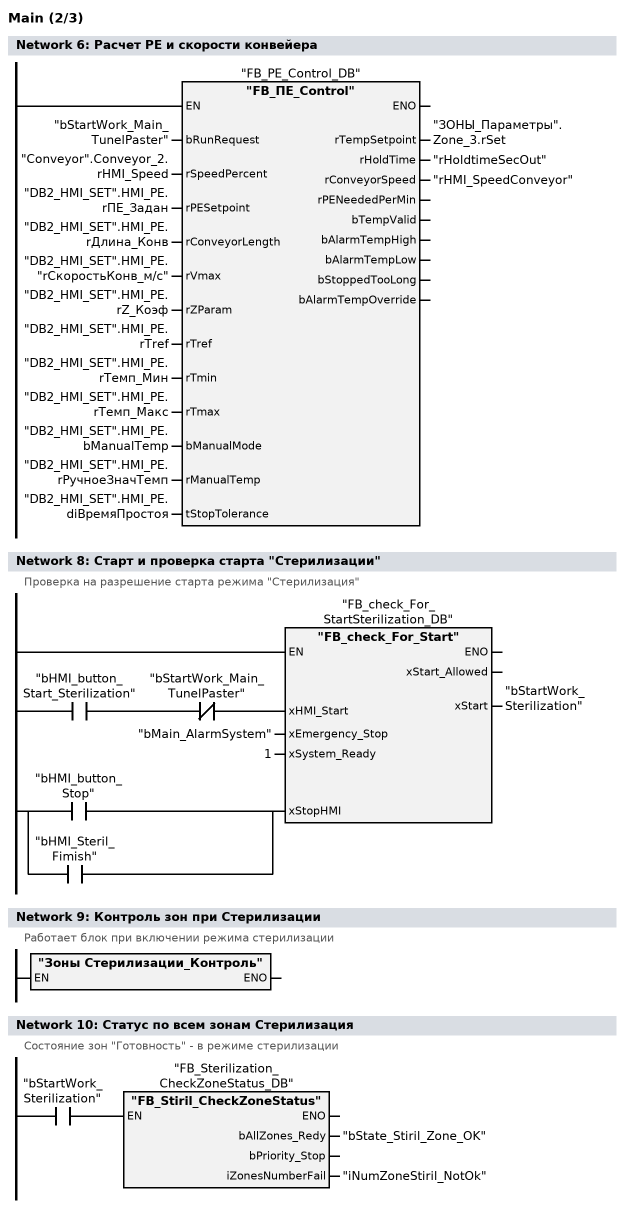
   RUNG wire#powerrail
      "FB_PE_Control_DB"(bRunRequest := "bStartWork_Main_TunelPaster", rSpeedPercent := "Conveyor".Conveyor_2.rHMI_Speed, rPESetpoint := "DB2_HMI_SET".HMI_PE.rПЕ_Задан, rConveyorLength := "DB2_HMI_SET".HMI_PE.rДлина_Конв, rVmax := "DB2_HMI_SET".HMI_PE."rСкоростьКонв_м/с", rZParam := "DB2_HMI_SET".HMI_PE.rZ_Коэф, rTref := "DB2_HMI_SET".HMI_PE.rТref, rTmin := "DB2_HMI_SET".HMI_PE.rТемп_Мин, rTmax := "DB2_HMI_SET".HMI_PE.rТемп_Макс, bManualMode := "DB2_HMI_SET".HMI_PE.bManualTemp, rManualTemp := "DB2_HMI_SET".HMI_PE.rРучноеЗначТемп, tStopTolerance := "DB2_HMI_SET".HMI_PE.diВремяПростоя, rTempSetpoint => "ЗОНЫ_Параметры".Zone_3.rSet, rHoldTime => "rHoldtimeSecOut", rConveyorSpeed => "rHMI_SpeedConveyor", rPENeededPerMin =>, bTempValid =>, bAlarmTempHigh =>, bAlarmTempLow =>, bStoppedTooLong =>, bAlarmTempOverride =>)
   END_RUNG
   // the same network as SCL:
   "FB_PE_Control_DB"(bRunRequest := "bStartWork_Main_TunelPaster",   // "FB_ПЕ_Control"
                      rSpeedPercent := "Conveyor".Conveyor_2.rHMI_Speed,
                      rPESetpoint := "DB2_HMI_SET".HMI_PE.rПЕ_Задан,
                      rConveyorLength := "DB2_HMI_SET".HMI_PE.rДлина_Конв,
                      rVmax := "DB2_HMI_SET".HMI_PE."rСкоростьКонв_м/с",
                      rZParam := "DB2_HMI_SET".HMI_PE.rZ_Коэф,
                      rTref := "DB2_HMI_SET".HMI_PE.rТref,
                      rTmin := "DB2_HMI_SET".HMI_PE.rТемп_Мин,
                      rTmax := "DB2_HMI_SET".HMI_PE.rТемп_Макс,
                      bManualMode := "DB2_HMI_SET".HMI_PE.bManualTemp,
                      rManualTemp := "DB2_HMI_SET".HMI_PE.rРучноеЗначТемп,
                      tStopTolerance := "DB2_HMI_SET".HMI_PE.diВремяПростоя,
                      rTempSetpoint => "ЗОНЫ_Параметры".Zone_3.rSet,
                      rHoldTime => "rHoldtimeSecOut",
                      rConveyorSpeed => "rHMI_SpeedConveyor");
END_REGION

REGION Network 7 (SCL): Перевод времени выдержки в минуты
   "rHMI_TimeHoldMin"  := "rHoldtimeSecOut" / 1;
   "rHMI_SpeedConveyor" := "rHMI_SpeedConveyor" * 1;
END_REGION

REGION Network 8: Старт и проверка старта "Стерилизации"
   // Проверка на разрешение старта режима "Стерилизация"
   RUNG wire#powerrail
      "FB_check_For_StartSterilization_DB"(xHMI_Start := wire#w1, xStopHMI := wire#w2, xEmergency_Stop := "bMain_AlarmSystem", xSystem_Ready := 1, xStart_Allowed =>, xStart => "bStartWork_Sterilization")
   END_RUNG
   RUNG wire#powerrail
      Contact( "bHMI_button_Start_Sterilization" )
      I_Contact( "bStartWork_Main_TunelPaster" )
   END_RUNG wire#w1
   RUNG wire#powerrail
      Contact( "bHMI_button_Stop" )
   END_RUNG wire#w2
   RUNG wire#powerrail
      Contact( "bHMI_Steril_Fimish" )
   END_RUNG wire#w2
   // the same network as SCL:
   "FB_check_For_StartSterilization_DB"(xHMI_Start := "bHMI_button_Start_Sterilization" AND NOT "bStartWork_Main_TunelPaster",   // "FB_check_For_Start"
                           xEmergency_Stop := "bMain_AlarmSystem",
                           xSystem_Ready := 1,
                           xStopHMI := "bHMI_button_Stop" OR "bHMI_Steril_Fimish",
                           xStart => "bStartWork_Sterilization");
END_REGION

REGION Network 9: Контроль зон при Стерилизации
   // Работает блок при включении режима стерилизации
   RUNG wire#powerrail
      "Зоны Стерилизации_Контроль"()
   END_RUNG
   // the same network as SCL:
   "Зоны Стерилизации_Контроль"();
END_REGION

REGION Network 10: Статус по всем зонам Стерилизация
   // Состояние зон "Готовность" - в режиме стерилизации
   RUNG wire#powerrail
      Contact( "bStartWork_Sterilization" )
      "FB_Sterilization_CheckZoneStatus_DB"(bAllZones_Redy => "bState_Stiril_Zone_OK", bPriority_Stop =>, iZonesNumberFail => "iNumZoneStiril_NotOk")
   END_RUNG
   // the same network as SCL:
   IF "bStartWork_Sterilization" THEN
       "FB_Sterilization_CheckZoneStatus_DB"(bAllZones_Redy => "bState_Stiril_Zone_OK",   // "FB_Stiril_CheckZoneStatus"
                               iZonesNumberFail => "iNumZoneStiril_NotOk");
   END_IF;
END_REGION

REGION Network 11: Таймер стерилизации
   // Отсчет времени стерилизации
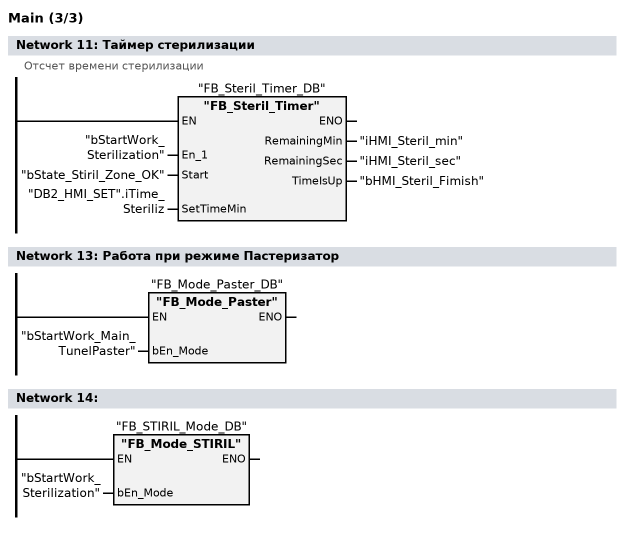
   RUNG wire#powerrail
      "FB_Steril_Timer_DB"(En_1 := "bStartWork_Sterilization", Start := "bState_Stiril_Zone_OK", SetTimeMin := "DB2_HMI_SET".iTime_Steriliz, RemainingMin => "iHMI_Steril_min", RemainingSec => "iHMI_Steril_sec", TimeIsUp => "bHMI_Steril_Fimish")
   END_RUNG
   // the same network as SCL:
   "FB_Steril_Timer_DB"(En_1 := "bStartWork_Sterilization",   // "FB_Steril_Timer"
                        Start := "bState_Stiril_Zone_OK",
                        SetTimeMin := "DB2_HMI_SET".iTime_Steriliz,
                        RemainingMin => "iHMI_Steril_min",
                        RemainingSec => "iHMI_Steril_sec",
                        TimeIsUp => "bHMI_Steril_Fimish");
END_REGION

REGION Network 12 (SCL): Окно окончания стирилизации
   IF "bHMI_Steril_Fimish" THEN
       "iHMIWind_FinishStiril" := 148;
   END_IF;
END_REGION

REGION Network 13: Работа при режиме Пастеризатор
   RUNG wire#powerrail
      "FB_Mode_Paster_DB"(bEn_Mode := "bStartWork_Main_TunelPaster")
   END_RUNG
   // the same network as SCL:
   "FB_Mode_Paster_DB"(bEn_Mode := "bStartWork_Main_TunelPaster");   // "FB_Mode_Paster"
END_REGION

REGION Network 14
   RUNG wire#powerrail
      "FB_STIRIL_Mode_DB"(bEn_Mode := "bStartWork_Sterilization")
   END_RUNG
   // the same network as SCL:
   "FB_STIRIL_Mode_DB"(bEn_Mode := "bStartWork_Sterilization");   // "FB_Mode_STIRIL"
END_REGION
END_ORGANIZATION_BLOCK

ORGANIZATION_BLOCK "PID"   // OB30, LAD, CyclicInterrupt
{ S7_Optimized_Access := 'TRUE' }
VERSION : 0.1
   VAR_INPUT
      Initial_Call : Bool;   // Initial call of this OB
      Event_Count : Int;   // Events discarded
   END_VAR
BEGIN

REGION Network 1: ПИД - Зона 1
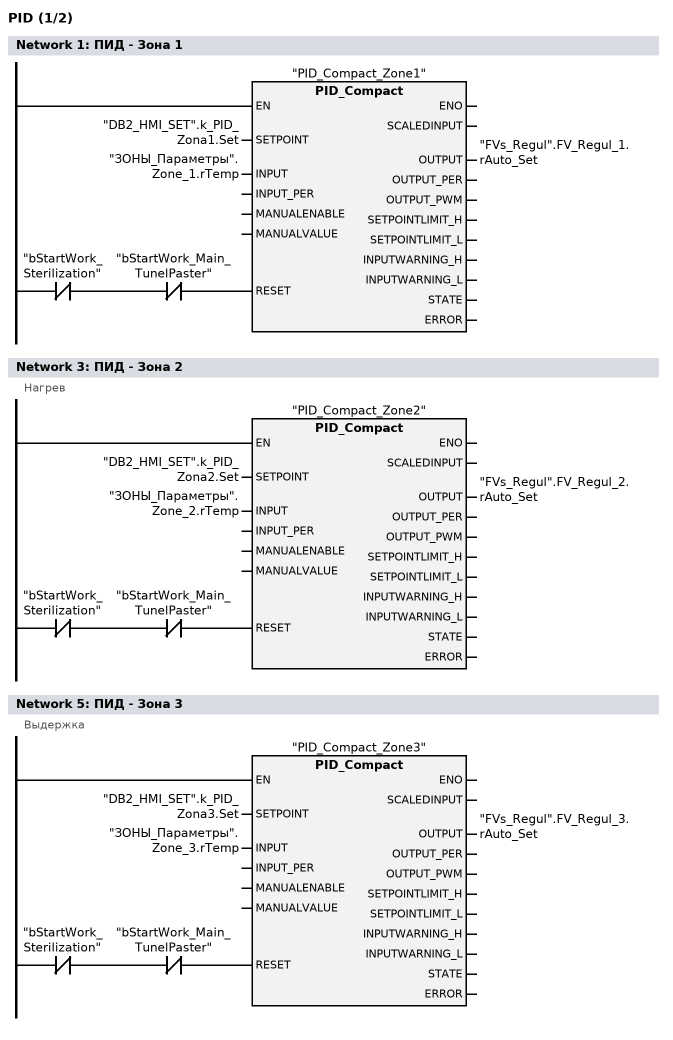
   "PID_Compact_Zone1"(Setpoint := "DB2_HMI_SET".k_PID_Zona1.Set,   // PID_Compact
                       Input := "ЗОНЫ_Параметры".Zone_1.rTemp,
                       Reset := NOT "bStartWork_Sterilization" AND NOT "bStartWork_Main_TunelPaster",
                       Output => "FVs_Regul".FV_Regul_1.rAuto_Set);
END_REGION

REGION Network 2 (SCL): Выбор типа ПИД - Зона 1
   //Режим работы ПИД - 0 - Нагрев; 1 - Охлаждение
   "PID_Compact_Zone1".sPid_Cmpt.b_InvCtrl := "bTypePID_Zone1";
   //Задание коэффициэнтов в ручном режиме

   "PID_Compact_Zone1".sRet.r_Ctrl_Gain := "DB2_HMI_SET".k_PID_Zona1.Gain; // Изменение коэф. П
   "PID_Compact_Zone1".sRet.r_Ctrl_Ti  := "DB2_HMI_SET".k_PID_Zona1.I; // Изменение коэф И
   "PID_Compact_Zone1".sRet.r_Ctrl_Td  := "DB2_HMI_SET".k_PID_Zona1.D; // Изменение коэф Д
END_REGION

REGION Network 3: ПИД - Зона 2
   // Нагрев
   "PID_Compact_Zone2"(Setpoint := "DB2_HMI_SET".k_PID_Zona2.Set,   // PID_Compact
                       Input := "ЗОНЫ_Параметры".Zone_2.rTemp,
                       Reset := NOT "bStartWork_Sterilization" AND NOT "bStartWork_Main_TunelPaster",
                       Output => "FVs_Regul".FV_Regul_2.rAuto_Set);
END_REGION

REGION Network 4 (SCL): Выбор типа ПИД Зона 2
   // 0 - Нагрев; 1 - Охлаждение
   "PID_Compact_Zone2".sPid_Cmpt.b_InvCtrl := "bTypePID_Zone2";
   //Задание коэффициэнтов в ручном режиме

   "PID_Compact_Zone2".sRet.r_Ctrl_Gain := "DB2_HMI_SET".k_PID_Zona2.Gain; // Изменение коэф. П
   "PID_Compact_Zone2".sRet.r_Ctrl_Ti := "DB2_HMI_SET".k_PID_Zona2.I; // Изменение коэф И
   "PID_Compact_Zone2".sRet.r_Ctrl_Td := "DB2_HMI_SET".k_PID_Zona2.D; // Изменение коэф Д
END_REGION

REGION Network 5: ПИД - Зона 3
   // Выдержка
   "PID_Compact_Zone3"(Setpoint := "DB2_HMI_SET".k_PID_Zona3.Set,   // PID_Compact
                       Input := "ЗОНЫ_Параметры".Zone_3.rTemp,
                       Reset := NOT "bStartWork_Sterilization" AND NOT "bStartWork_Main_TunelPaster",
                       Output => "FVs_Regul".FV_Regul_3.rAuto_Set);
END_REGION

REGION Network 6 (SCL): Выбор типа ПИД Зона 3
   // 0 - Нагрев; 1 - Охлаждение
   "PID_Compact_Zone3".sPid_Cmpt.b_InvCtrl := "bTypePID_Zone3";
   //Задание коэффициэнтов в ручном режиме
   "PID_Compact_Zone3".sRet.r_Ctrl_Gain := "DB2_HMI_SET".k_PID_Zona3.Gain; // Изменение коэф. П
   "PID_Compact_Zone3".sRet.r_Ctrl_Ti :=   "DB2_HMI_SET".k_PID_Zona3.I;    // Изменение коэф И
   "PID_Compact_Zone3".sRet.r_Ctrl_Td :=   "DB2_HMI_SET".k_PID_Zona3.D;    // Изменение коэф Д
END_REGION

REGION Network 7: ПИД - Зона 4
   // Выдержка
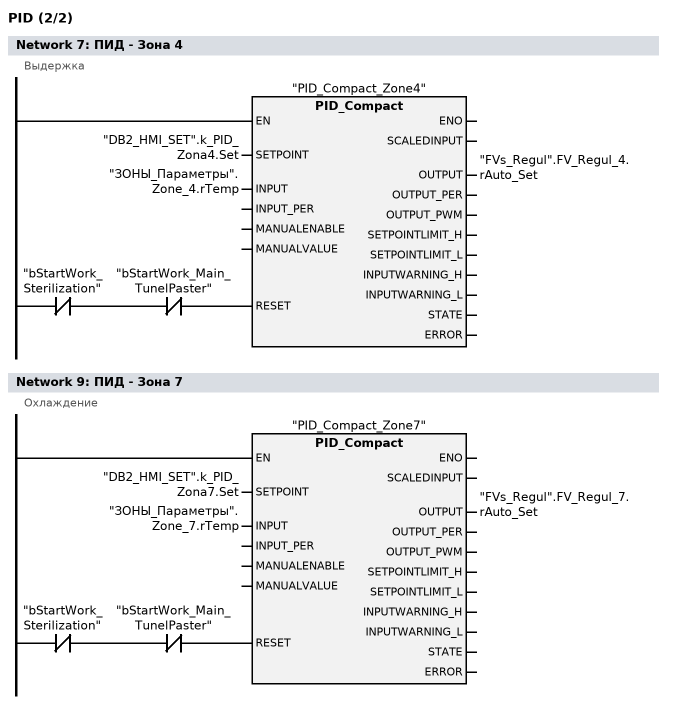
   "PID_Compact_Zone4"(Setpoint := "DB2_HMI_SET".k_PID_Zona4.Set,   // PID_Compact
                       Input := "ЗОНЫ_Параметры".Zone_4.rTemp,
                       Reset := NOT "bStartWork_Sterilization" AND NOT "bStartWork_Main_TunelPaster",
                       Output => "FVs_Regul".FV_Regul_4.rAuto_Set);
END_REGION

REGION Network 8 (SCL): Выбор типа ПИД Зона 4
   // 0 - Нагрев; 1 - Охлаждение
   "PID_Compact_Zone4".sPid_Cmpt.b_InvCtrl := TRUE;
   //Задание коэффициэнтов в ручном режиме
   "PID_Compact_Zone4".sRet.r_Ctrl_Gain := "DB2_HMI_SET".k_PID_Zona4.Gain; // Изменение коэф. П
   "PID_Compact_Zone4".sRet.r_Ctrl_Ti := "DB2_HMI_SET".k_PID_Zona4.I;    // Изменение коэф И
   "PID_Compact_Zone4".sRet.r_Ctrl_Td := "DB2_HMI_SET".k_PID_Zona4.D;    // Изменение коэф Д
END_REGION

REGION Network 9: ПИД - Зона 7
   // Охлаждение
   "PID_Compact_Zone7"(Setpoint := "DB2_HMI_SET".k_PID_Zona7.Set,   // PID_Compact
                       Input := "ЗОНЫ_Параметры".Zone_7.rTemp,
                       Reset := NOT "bStartWork_Sterilization" AND NOT "bStartWork_Main_TunelPaster",
                       Output => "FVs_Regul".FV_Regul_7.rAuto_Set);
END_REGION

REGION Network 10 (SCL): Выбор типа ПИД Зона 7
   // 0 - Нагрев; 1 - Охлаждение
   "PID_Compact_Zone7".sPid_Cmpt.b_InvCtrl := TRUE;
   //Задание коэффициэнтов в ручном режиме
   "PID_Compact_Zone7".sRet.r_Ctrl_Gain := "DB2_HMI_SET".k_PID_Zona7.Gain; // Изменение коэф. П
   "PID_Compact_Zone7".sRet.r_Ctrl_Ti := "DB2_HMI_SET".k_PID_Zona7.I;      // Изменение коэф И
   "PID_Compact_Zone7".sRet.r_Ctrl_Td := "DB2_HMI_SET".k_PID_Zona7.D;      // Изменение коэф Д
END_REGION
END_ORGANIZATION_BLOCK

ORGANIZATION_BLOCK "Startup"   // OB100, SCL, Startup
TITLE = "Complete Restart"
{ S7_Optimized_Access := 'TRUE' }
VERSION : 0.1
   VAR_INPUT
      LostRetentive : Bool;   // True if retentive data are lost
      LostRTC : Bool;   // True if date and time are lost
   END_VAR
BEGIN
   "PID_Compact_Zone1".sRet.r_Ctrl_Gain := "PID_Compact_Zone1".sBackUp.r_Gain;
END_ORGANIZATION_BLOCK

ORGANIZATION_BLOCK "Исполнительные устройств"   // OB123, LAD, ProgramCycle
TITLE = Работа физических устройств
{ S7_Optimized_Access := 'TRUE' }
VERSION : 0.1
// Насосы, клапана, и т.д.
   VAR_INPUT
      Initial_Call : Bool;   // Initial call of this OB
      Remanence : Bool;   // =True, if remanent data are available
   END_VAR
BEGIN

REGION Network 1: Аналогвые датчики
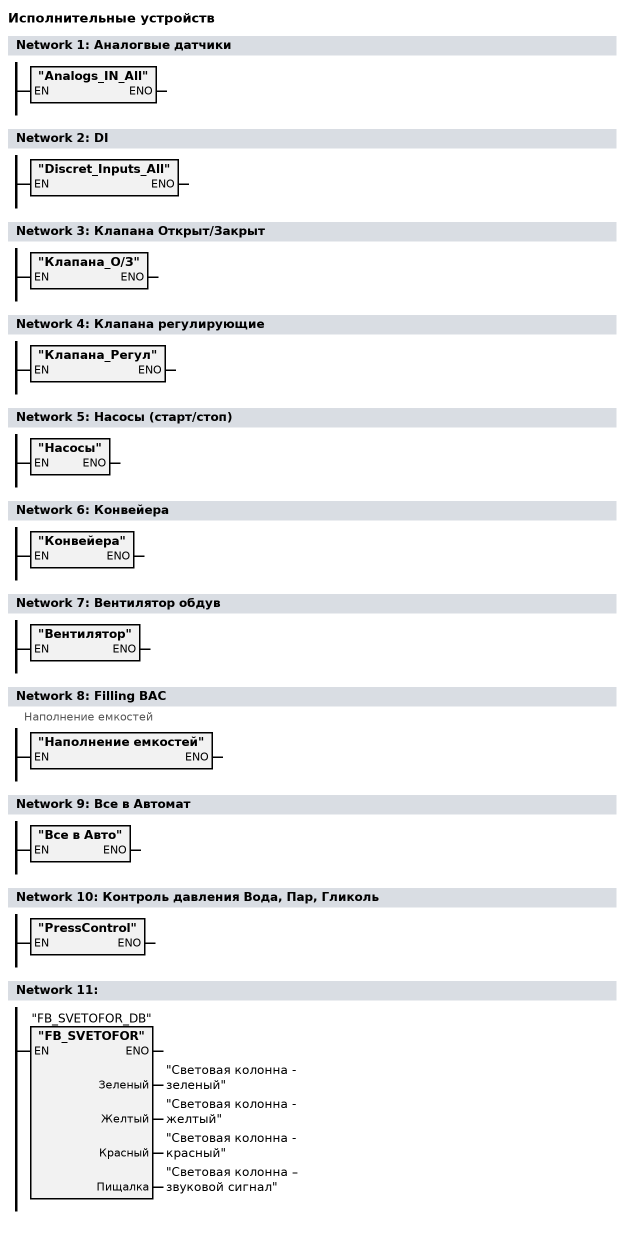
   RUNG wire#powerrail
      "Analogs_IN_All"()
   END_RUNG
   // the same network as SCL:
   "Analogs_IN_All"();
END_REGION

REGION Network 2: DI
   RUNG wire#powerrail
      "Discret_Inputs_All"()
   END_RUNG
   // the same network as SCL:
   "Discret_Inputs_All"();
END_REGION

REGION Network 3: Клапана Открыт/Закрыт
   RUNG wire#powerrail
      "Клапана_О/З"()
   END_RUNG
   // the same network as SCL:
   "Клапана_О/З"();
END_REGION

REGION Network 4: Клапана регулирующие
   RUNG wire#powerrail
      "Клапана_Регул"()
   END_RUNG
   // the same network as SCL:
   "Клапана_Регул"();
END_REGION

REGION Network 5: Насосы (старт/стоп)
   RUNG wire#powerrail
      "Насосы"()
   END_RUNG
   // the same network as SCL:
   "Насосы"();
END_REGION

REGION Network 6: Конвейера
   RUNG wire#powerrail
      "Конвейера"()
   END_RUNG
   // the same network as SCL:
   "Конвейера"();
END_REGION

REGION Network 7: Вентилятор обдув
   RUNG wire#powerrail
      "Вентилятор"()
   END_RUNG
   // the same network as SCL:
   "Вентилятор"();
END_REGION

REGION Network 8: Filling BAC
   // Наполнение емкостей
   RUNG wire#powerrail
      "Наполнение емкостей"()
   END_RUNG
   // the same network as SCL:
   "Наполнение емкостей"();
END_REGION

REGION Network 9: Все в Автомат
   RUNG wire#powerrail
      "Все в Авто"()
   END_RUNG
   // the same network as SCL:
   "Все в Авто"();
END_REGION

REGION Network 10: Контроль давления Вода, Пар, Гликоль
   RUNG wire#powerrail
      "PressControl"()
   END_RUNG
   // the same network as SCL:
   "PressControl"();
END_REGION

REGION Network 11
   RUNG wire#powerrail
      "FB_SVETOFOR_DB"(Зеленый => "Световая колонна - зеленый", Желтый => "Световая колонна - желтый", Красный => "Световая колонна - красный", Пищалка => "Световая колонна – звуковой сигнал")
   END_RUNG
   // the same network as SCL:
   "FB_SVETOFOR_DB"(Зеленый => "Световая колонна - зеленый",   // "FB_SVETOFOR"
                    Желтый => "Световая колонна - желтый",
                    Красный => "Световая колонна - красный",
                    Пищалка => "Световая колонна – звуковой сигнал");
END_REGION
END_ORGANIZATION_BLOCK

// folder: AI_Signal

FUNCTION_BLOCK "AI_(4-20)_1"   // FB13, LAD
{ S7_Optimized_Access := 'FALSE' }
VERSION : 0.1
   VAR_INPUT
      Input_PLC : Int;   // Вход_Значение на ПЛК
      "HMI_Simulate_on/off" : Bool;   // 0 - выкл, 1 - вкл
      HMI_rSimulate_value : Real;   // значение
      HMI_rParam_Sensor_HL : Real := 16.0;   // Параметры датчика по паспорту (макс значение)bar, C, итд
      HMI_rParam_Sensor_LL : Real;   // Параметры датчика по паспорту (мин значение)bar, C, итд
      "HMI_Filtr_On/off" : Bool;   // Фильтрация, true - вкл
   END_VAR
   VAR_OUTPUT
      Error_out : Bool;   // Ошибка датчика
      HMI_Value_OUT : Real;   // Значение в ед. измерения
   END_VAR
   VAR
      OUT_Scale : Real;   // Выход скалированного значения
      OUT_Normal_Ed : Real;   // Выход нормализованной единицы от 0 др 1
      AI_filtr : "AI_Filtr";
      HMI_Range : Int := 10;   // Кол-во данных для фильтрации
      HMI_iSet_Tik : Int := 2;   // Скорость набора данных для фильтрации
   END_VAR
   VAR_TEMP
      Input_PLC_to_dint : DInt;   // Конвертация из инт в реал
      Error : Word;   // Ошибка в скалировании
      "PLC to_real" : Real;
      value_scale : Real;
      Input_PLC_temp : Int;
      OFF_Param : Bool;
   END_VAR
BEGIN

REGION Network 1
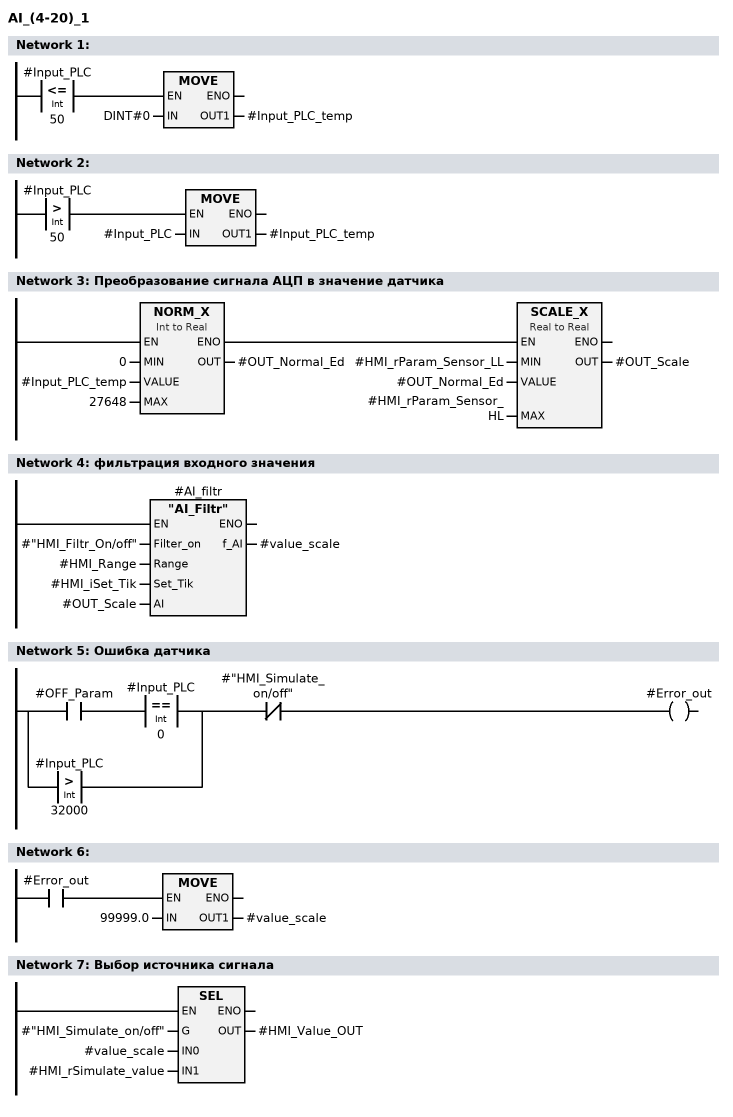
   RUNG wire#powerrail
      { S7_Templates := "SrcType := Int" } LE_Contact(in1 := #Input_PLC, in2 := 50)
      { S7_GenerateENO := "TRUE" } Move(in := DINT#0, out1 => #Input_PLC_temp)
   END_RUNG
   // the same network as SCL:
   IF #Input_PLC <= 50 THEN #Input_PLC_temp := DINT#0; END_IF;
END_REGION

REGION Network 2
   RUNG wire#powerrail
      { S7_Templates := "SrcType := Int" } GT_Contact(in1 := #Input_PLC, in2 := 50)
      { S7_GenerateENO := "TRUE" } Move(in := #Input_PLC, out1 => #Input_PLC_temp)
   END_RUNG
   // the same network as SCL:
   IF #Input_PLC > 50 THEN #Input_PLC_temp := #Input_PLC; END_IF;
END_REGION

REGION Network 3: Преобразование сигнала АЦП в значение датчика
   RUNG wire#powerrail
      { S7_Templates := "[SrcType := Int, DestType := Real]" } Normalize(min := 0, value := #Input_PLC_temp, max := 27648, out => #OUT_Normal_Ed)
      { S7_Templates := "[SrcType := Real, DestType := Real]" } Scale(min := #HMI_rParam_Sensor_LL, value := #OUT_Normal_Ed, max := #HMI_rParam_Sensor_HL, out => #OUT_Scale)
   END_RUNG
   // the same network as SCL:
   #OUT_Normal_Ed := NORM_X(MIN := 0, VALUE := #Input_PLC_temp, MAX := 27648);
   #OUT_Scale := SCALE_X(MIN := #HMI_rParam_Sensor_LL, VALUE := #OUT_Normal_Ed, MAX := #HMI_rParam_Sensor_HL);
END_REGION

REGION Network 4: фильтрация входного значения
   RUNG wire#powerrail
      #AI_filtr(Filter_on := #"HMI_Filtr_On/off", Range := #HMI_Range, Set_Tik := #HMI_iSet_Tik, AI := #OUT_Scale, f_AI => #value_scale)
   END_RUNG
   // the same network as SCL:
   #AI_filtr(Filter_on := #"HMI_Filtr_On/off",   // "AI_Filtr"
             Range := #HMI_Range,
             Set_Tik := #HMI_iSet_Tik,
             AI := #OUT_Scale,
             f_AI => #value_scale);
END_REGION

REGION Network 5: Ошибка датчика
   RUNG wire#powerrail
      Contact( #OFF_Param )
      { S7_Templates := "SrcType := Int" } EQ_Contact(in1 := #Input_PLC, in2 := 0)
      wire#w1
      I_Contact( #"HMI_Simulate_on/off" )
      Coil( #Error_out )
   END_RUNG
   RUNG wire#powerrail
      { S7_Templates := "SrcType := Int" } GT_Contact(in1 := #Input_PLC, in2 := 32000)
   END_RUNG wire#w1
   // the same network as SCL:
   #Error_out := ((#OFF_Param AND (#Input_PLC = 0)) OR (#Input_PLC > 32000)) AND NOT #"HMI_Simulate_on/off";
END_REGION

REGION Network 6
   RUNG wire#powerrail
      Contact( #Error_out )
      Move(in := 99999.0, out1 => #value_scale)
   END_RUNG
   // the same network as SCL:
   IF #Error_out THEN #value_scale := 99999.0; END_IF;
END_REGION

REGION Network 7: Выбор источника сигнала
   #HMI_Value_OUT := SEL(G := #"HMI_Simulate_on/off", IN0 := #value_scale, IN1 := #HMI_rSimulate_value);
END_REGION
END_FUNCTION_BLOCK

FUNCTION_BLOCK "AI_(PT100)"   // FB21, LAD
{ S7_Optimized_Access := 'FALSE' }
VERSION : 0.1
   VAR_INPUT
      Input_PLC : Int;   // Вход_Значение на ПЛК
      "Simulate_on/off" : Bool;   // 0 - выкл, 1 - вкл
      Simulate_value : Real;   // значение
      Param_Sensor_HL : Real := 16.0;   // Параметры датчика по паспорту (макс значение)bar, C, итд
      Param_Sensor_LL : Real;   // Параметры датчика по паспорту (мин значение)bar, C, итд
      "Filtr_On/off" : Bool;   // Фильтрация, true - вкл
   END_VAR
   VAR_OUTPUT
      Value_OUT : Real;   // Значение в ед. измерения
      Error_out : Bool;   // Ошибка датчика
   END_VAR
   VAR
      bipolar : Bool;
      OUT_Scale : Real;   // Выход скалированного значения
      AI_filtr : "AI_Filtr";
      Range : Int := 10;   // Кол-во данных для фильтрации
   END_VAR
   VAR_TEMP
      Input_PLC_to_dint : DInt;   // Конвертация из инт в реал
      Error : Word;   // Ошибка в скалировании
      "PLC to_real" : Real;
      value_scale : Real;
      Input_PLC_temp : Int;
      Input_PLC_to_real : Real;
   END_VAR
BEGIN

REGION Network 1
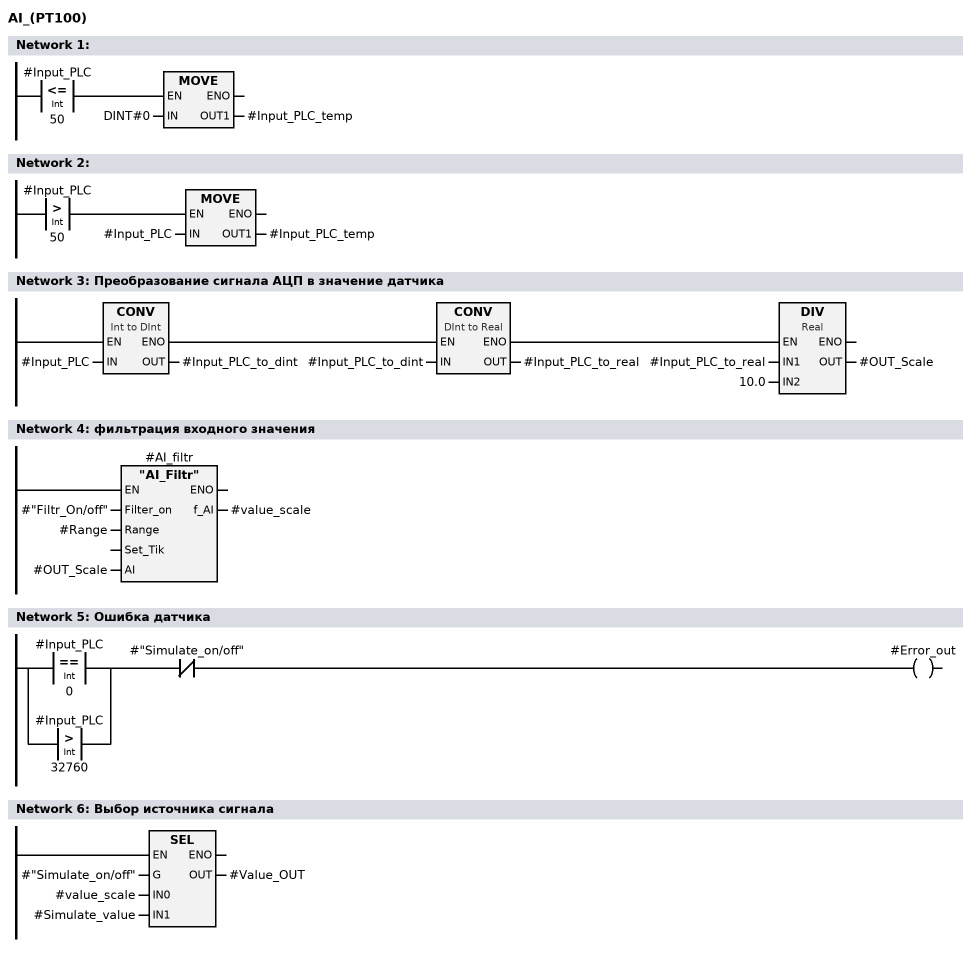
   RUNG wire#powerrail
      { S7_Templates := "SrcType := Int" } LE_Contact(in1 := #Input_PLC, in2 := 50)
      { S7_GenerateENO := "TRUE" } Move(in := DINT#0, out1 => #Input_PLC_temp)
   END_RUNG
   // the same network as SCL:
   IF #Input_PLC <= 50 THEN #Input_PLC_temp := DINT#0; END_IF;
END_REGION

REGION Network 2
   RUNG wire#powerrail
      { S7_Templates := "SrcType := Int" } GT_Contact(in1 := #Input_PLC, in2 := 50)
      { S7_GenerateENO := "TRUE" } Move(in := #Input_PLC, out1 => #Input_PLC_temp)
   END_RUNG
   // the same network as SCL:
   IF #Input_PLC > 50 THEN #Input_PLC_temp := #Input_PLC; END_IF;
END_REGION

REGION Network 3: Преобразование сигнала АЦП в значение датчика
   RUNG wire#powerrail
      { S7_Templates := "[SrcType := Int, DestType := DInt]"; S7_GenerateENO := "TRUE" } Convert(in := #Input_PLC, out => #Input_PLC_to_dint)
      { S7_Templates := "[SrcType := DInt, DestType := Real]"; S7_GenerateENO := "TRUE" } Convert(in := #Input_PLC_to_dint, out => #Input_PLC_to_real)
      { S7_Templates := "SrcType := Real"; S7_GenerateENO := "TRUE" } Div(in1 := #Input_PLC_to_real, in2 := 10.0, out => #OUT_Scale)
   END_RUNG
   // the same network as SCL:
   // ENO of a box is taken as its EN; it also drops when the box reports an error
   #Input_PLC_to_dint := INT_TO_DINT(#Input_PLC);
   #Input_PLC_to_real := DINT_TO_REAL(#Input_PLC_to_dint);
   #OUT_Scale := #Input_PLC_to_real / 10.0;
END_REGION

REGION Network 4: фильтрация входного значения
   RUNG wire#powerrail
      #AI_filtr(Filter_on := #"Filtr_On/off", Range := #Range, Set_Tik :=, AI := #OUT_Scale, f_AI => #value_scale)
   END_RUNG
   // the same network as SCL:
   #AI_filtr(Filter_on := #"Filtr_On/off", Range := #Range, AI := #OUT_Scale, f_AI => #value_scale);   // "AI_Filtr"
END_REGION

REGION Network 5: Ошибка датчика
   RUNG wire#powerrail
      { S7_Templates := "SrcType := Int" } EQ_Contact(in1 := #Input_PLC, in2 := 0)
      wire#w1
      I_Contact( #"Simulate_on/off" )
      Coil( #Error_out )
   END_RUNG
   RUNG wire#powerrail
      { S7_Templates := "SrcType := Int" } GT_Contact(in1 := #Input_PLC, in2 := 32760)
   END_RUNG wire#w1
   // the same network as SCL:
   #Error_out := ((#Input_PLC = 0) OR (#Input_PLC > 32760)) AND NOT #"Simulate_on/off";
END_REGION

REGION Network 6: Выбор источника сигнала
   #Value_OUT := SEL(G := #"Simulate_on/off", IN0 := #value_scale, IN1 := #Simulate_value);
END_REGION
END_FUNCTION_BLOCK

// folder: AI_Signal/Funktion

FUNCTION_BLOCK "AI_Filtr"   // FB14, SCL
{ S7_Optimized_Access := 'FALSE' }
VERSION : 0.1
   VAR_INPUT
      Filter_on : Bool;   // Вкл фильтрации
      Range : Int := 10;   // Кол-во входных значений для вычисления среднего
      Set_Tik : Int := 2;   // Задача периода фильтрации от 1(мин) до 8
      AI : Real;   // Вход значения датчика
   END_VAR
   VAR_OUTPUT
      f_AI : Real;   // выход значения с фильтром или без
   END_VAR
   VAR
      CTU : CTU_INT;   // счетчик для подсчета кол-во вх значений
      Tik : Bool;   // Время фильтрации
      ai_array : Array[0..#Max_Array] of Real;   // Массив значений датчика
      i : Int;   // для цикла ФОР
      sum_AI : Real;   // Суммирование значений с входа датчика
      Avarage_AI : Real;   // Среднее значение датчика
      fRS_set : Bool;   // Для RS тригера
      fRS_res : Bool;   // Для RS тригера
      fRS_out : Bool;   // Для RS тригера
      FullFiltr : Bool;   // Ожидание наполнения значений для вычисления средней
      Res_count : Bool;   // сброс счетчика
   END_VAR
   VAR CONSTANT
      Max_Array : Int := 30;   // Размер массива
   END_VAR
BEGIN

   CASE #Set_Tik OF                   
       1:  
           #Tik := "Time_0.1s";
       2:  
           #Tik := "Time_0.2s";
       3:
           #Tik := "Time_0.4s";
       4:
           #Tik := "Time_0.5s";
       5:
           #Tik := "Time_0.8s";
       6:
           #Tik := "Time_1s";
       7:
           #Tik := "Time_1.6s";
       8:
           #Tik := "Time_2s";
       0:
           #Tik := "Time_0.1s";

       ELSE  
           #Set_Tik := 8;
   END_CASE;  // Выбор периода фильтрации входного сигнала
   REGION RS триггер
       IF #fRS_set THEN
           #fRS_out := true;
       ELSIF #fRS_res AND NOT #fRS_set THEN
           #fRS_out := false;
       END_IF;
   END_REGION

   REGION Подсчет среднего значения входа
       // Statement section REGION
           #CTU(CU := #Tik,
                PV := #Range,
                R := #Res_count,
                Q => #Res_count);                                      // Счетчик для набора значений с входа
           #ai_array[#CTU.CV] := #AI;                                  // Запись значений с входа в массив

           IF #Res_count THEN                                              // СБРОС как счетчик переполниться Для корректной работы счетчика
               #i := 0;
               #sum_AI := 0;
           END_IF;

           IF #Range <> #i THEN                                    // выход из цикла FOR при суммировании всех значений, почему то сам не прекращел подсчет при окончании цикла все время суммировался 
               FOR #i := 0 TO (#Range - 1) DO
                   #sum_AI := #ai_array[#i] + #sum_AI;             // суммирование значений
               END_FOR;
           END_IF;

       #Avarage_AI := #sum_AI / #Range;                             // Вычисление среднего значения
       #fRS_res := NOT #Filter_on;

   END_REGION

   REGION Выбор выхода прямое или фильтрованное значение
       IF #Filter_on THEN                                          //Включение выключение фильтрации
           #fRS_set := #CTU.QD;                                    //При включении фильтра ждем наполнения значениями с входа, пока ждем - отправляем на выход прямое значение входа, далее фильтруем
            #FullFiltr := #fRS_out;

          IF #FullFiltr THEN                                       //Когда фильтр наполнился - вывыодим среднее значение входа
               #f_AI := #Avarage_AI;                              // ЗАпись значения на выход AI
          ELSE
               #f_AI := #AI;                                     // Прямой вывод значения, пока значения не наполнились данными
          END_IF;
       ELSE
           #f_AI := #AI;                                        // Если фильтр выключен, на выход прямое значение с входа
       END_IF; 

   END_REGION
END_FUNCTION_BLOCK

FUNCTION "Calculate_AI" : Void   // FC7, SCL
{ S7_Optimized_Access := 'FALSE' }
VERSION : 0.1
   VAR_INPUT
      IN_sensors : Int;
      Current_max : Real;
      Current_min : Real;
      Code_HL : Real;
      Code_LL : Real;
      Param_Sensor_HL : Real;   // Параметры датчика по паспорту (макс значение)bar, C, итд
      Param_Sensor_LL : Real;   // Параметры датчика по паспорту (мин значение)bar, C, итд
   END_VAR
   VAR_OUTPUT
      signal_Electric : Real;   // выход в электрических ед измерения
      Value_Sensor : Real;   // выход реального значения датчика в ед измерения
   END_VAR
   VAR_TEMP
      sensor_to_real : Real;   // Для конвертации INT to Real
      result_to_out_signal : Real;   // Для вычитания реального значения показания датчика
   END_VAR
BEGIN
       //Convert int to real
   #sensor_to_real := INT_TO_REAL(#IN_sensors);

       // Расчет значения АЦП контроллера в значение эл. ед измерения (I, U) в зависимости от значений на входе
   #signal_Electric := ((#sensor_to_real - #Code_LL) * (#Current_max - #Current_min) / (#Code_HL - #Code_LL))+ #Current_min;
   #result_to_out_signal := #signal_Electric;

   // Расчет значения в реальных единицах измерения датчика (bar, C,) в зависимости от введеных параметров датчика Param_Sensor min/max
   #Value_Sensor := (#result_to_out_signal - #Current_min) * (#Param_Sensor_HL - #Param_Sensor_LL) / (#Current_max - #Current_min) + #Param_Sensor_LL;
END_FUNCTION

// folder: DI_signal

FUNCTION_BLOCK "FB_DI"   // FB15, LAD
TITLE = Блок обработки дискретных входов
{ S7_Optimized_Access := 'FALSE' }
VERSION : 0.1
   VAR_INPUT
      input_value : Bool;   // Входной тэг контроллера
      "On/Off_Filters_DI" : Bool;   // Вкл/выкл фильтрацию входа
      Set_Time_Dely : Time;   // Уставка времени фильтрации
      Simulate : Bool;   // Симуляция входа (Вкл/Выкл)
      Simulate_Value : Bool;   // Значение симуляции
   END_VAR
   VAR_OUTPUT
      Value : Bool;   // Обработанный сигнал
   END_VAR
   VAR
      Time_Delay : Time;   // Время фильтрации для таймера
      Time_On : TON_TIME;   // Фильтр на Вкл
      Time_Off : TON_TIME;   // Фильтр на Выкл
      Nul_Time : Time := T#1MS;   // Откл фильтрации (0)
   END_VAR
BEGIN

REGION Network 1: Включение фильтрации
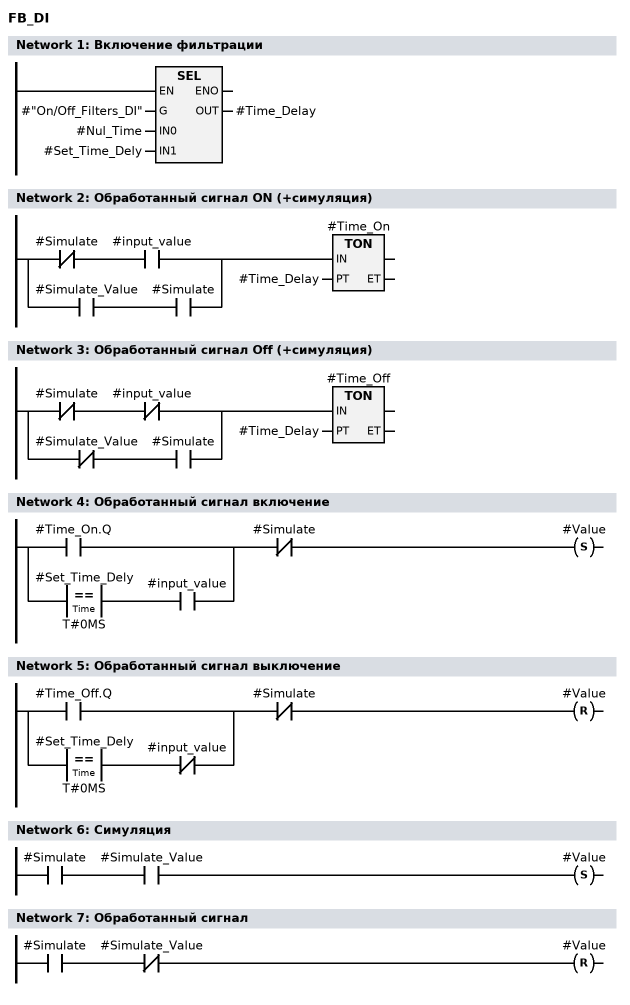
   #Time_Delay := SEL(G := #"On/Off_Filters_DI", IN0 := #Nul_Time, IN1 := #Set_Time_Dely);
END_REGION

REGION Network 2: Обработанный сигнал ON (+симуляция)
   #Time_On(IN := (NOT #Simulate AND #input_value) OR (#Simulate_Value AND #Simulate), PT := #Time_Delay);   // TON
END_REGION

REGION Network 3: Обработанный сигнал Off (+симуляция)
   #Time_Off(IN := (NOT #Simulate AND NOT #input_value) OR (NOT #Simulate_Value AND #Simulate),   // TON
             PT := #Time_Delay);
END_REGION

REGION Network 4: Обработанный сигнал включение
   RUNG wire#powerrail
      Contact( #Time_On.Q )
      wire#w1
      I_Contact( #Simulate )
      S_Coil( #Value )
   END_RUNG
   RUNG wire#powerrail
      { S7_Templates := "SrcType := Time" } EQ_Contact(in1 := #Set_Time_Dely, in2 := T#0MS)
      Contact( #input_value )
   END_RUNG wire#w1
   // the same network as SCL:
   IF (#Time_On.Q OR ((#Set_Time_Dely = T#0MS) AND #input_value)) AND NOT #Simulate THEN
       #Value := TRUE;
   END_IF;
END_REGION

REGION Network 5: Обработанный сигнал выключение
   RUNG wire#powerrail
      Contact( #Time_Off.Q )
      wire#w1
      I_Contact( #Simulate )
      R_Coil( #Value )
   END_RUNG
   RUNG wire#powerrail
      { S7_Templates := "SrcType := Time" } EQ_Contact(in1 := #Set_Time_Dely, in2 := T#0MS)
      I_Contact( #input_value )
   END_RUNG wire#w1
   // the same network as SCL:
   IF (#Time_Off.Q OR ((#Set_Time_Dely = T#0MS) AND NOT #input_value)) AND NOT #Simulate THEN
       #Value := FALSE;
   END_IF;
END_REGION

REGION Network 6: Симуляция
   RUNG wire#powerrail
      Contact( #Simulate )
      Contact( #Simulate_Value )
      S_Coil( #Value )
   END_RUNG
   // the same network as SCL:
   IF #Simulate AND #Simulate_Value THEN #Value := TRUE; END_IF;
END_REGION

REGION Network 7: Обработанный сигнал
   RUNG wire#powerrail
      Contact( #Simulate )
      I_Contact( #Simulate_Value )
      R_Coil( #Value )
   END_RUNG
   // the same network as SCL:
   IF #Simulate AND NOT #Simulate_Value THEN #Value := FALSE; END_IF;
END_REGION
END_FUNCTION_BLOCK

// folder: FB

FUNCTION_BLOCK "R_trig"   // FB16, SCL
{ S7_Optimized_Access := 'TRUE' }
VERSION : 0.1
   VAR_INPUT
      In : Bool;
   END_VAR
   VAR_OUTPUT
      Q : Bool;
   END_VAR
   VAR
      Click_M : Bool;
   END_VAR
BEGIN
   #Q := #In AND NOT #Click_M;
   #Click_M := #In;
END_FUNCTION_BLOCK